RoboDK station: Implementación.rdk

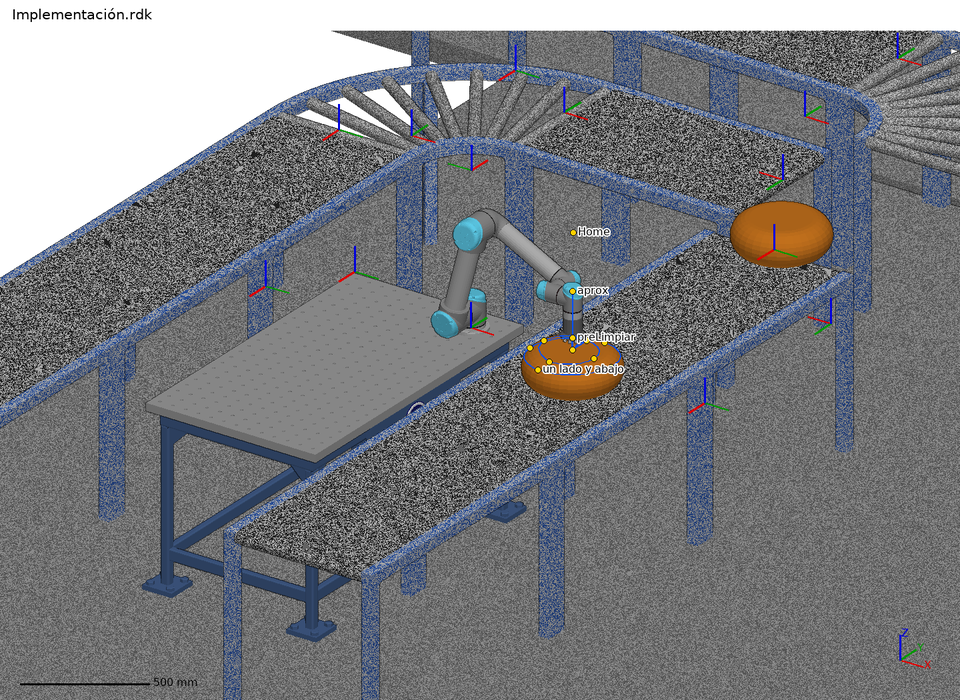
[picture v0: the station drawn from its stored meshes, robots at their saved joint values, targets as dots, program paths as lines]
Station Implementación (saved by RoboDK 5.8.0). Poses are relative to the parent item; angles as X-Y-Z fixed-axis rotations.
  - object Base UR20e at (0, 0, 0) mm, size 250 x 250 x 500 mm, geometry from LayOut general robodk v7 3.step
  - object Suelo at (0, 0, 0) mm, size 13800 x 12750 x 101 mm, geometry from LayOut general robodk v7.step
  - object Estater at (0, 0, 0) mm, size 1550 x 550 x 2250 mm, geometry from LayOut general robodk v7 2.step
  - frame Esquina implantación at (-4000, -50, 1) mm, rotated rx 0 ry 0 rz -90 deg
    - frame mesaRobots at (3150, 1450, 800) mm
      - object mesa at (350, 400, 0) mm, size 1420 x 820 x 800 mm, geometry from Table-1400x800x800mm.sld
      - object keso at (250, 1075, -50) mm, size 400 x 400 x 150 mm, geometry from Queso v10.step
      - frame UR5 Base at (150, 650, 0) mm, rotated rx 0 ry 0 rz 90 deg
        - robot UR5: 6 axes
            modified DH rows (alpha deg, a mm, theta deg, d mm): 0, 0, 0, 89.2; 90, 0, 180, 0; 0, 425, 0, 0; 0, 392, 0, 109.3; -90, 0, 0, 94.75; 90, 0, 180, 82.5
            joint limits [-360, -360, -360, -360, -360, -360] to [360, 360, 360, 360, 360, 360]; home [0, -90, -90, 0, 90, 0]; saved at [0.97, -104.431, -103.116, -62.453, 90, 0.97]
          - tool HerramientaCepillo v3 v3, TCP at (0, 0, 87) mm, size 103 x 102.7 x 101.3 mm, geometry from HerramientaCepillo v3 v3.step
        - target Home (Cartesian target) at (561.5, -109.3, 608.95) mm, rotated rx -90 ry 0 rz -90 deg; joints [0, -90, -90, 0, 90, 0] of UR5
        - target aprox (Cartesian target) at (550, -100, 350) mm, rotated rx 180 ry 0 rz -90 deg; joints [0.97, -98.334, -80.235, -91.431, 90, 0.97] of UR5
        - target preLimpiar (Cartesian target) at (550, -100, 150) mm, rotated rx 180 ry 0 rz -90 deg; joints [158.42, -51.501, -293.37, -285.129, 90, 158.42] of UR5
        - target contactoQueso (Cartesian target) at (550, -100, 100) mm, rotated rx 180 ry 0 rz -90 deg; joints [0.97, -108.044, -106.77, -55.186, 90, 0.97] of UR5
        - target cerca y abajo (Cartesian target) at (362.36, -117.41, 62.97) mm, rotated rx -122.07 ry 2.25 rz -86.41 deg; joints [-5.256, -118.006, -154.949, 60.494, 98.681, -2.826] of UR5
        - target un lado y abajo (Cartesian target) at (510.77, -278.06, 72.55) mm, rotated rx -157.33 ry 40.11 rz -72.05 deg; joints [-29.262, -119.839, -98.457, -65.594, 133.363, -44.391] of UR5
        - target lejos y abajo (Cartesian target) at (730.3, -97.43, 74.87) mm, rotated rx 141.57 ry 25.71 rz -56.33 deg; joints [1.508, -156.051, -23.971, -135.034, 87.527, -40.229] of UR5
        - target otro lado y abajo (Cartesian target) at (570.65, 88.54, 61.08) mm, rotated rx 122.05 ry -0.47 rz -5.3 deg; joints [31.697, -122.988, -92.801, -97.883, 47.184, -34.887] of UR5
        - target cerca (Cartesian target) at (413.04, -94.57, 98.6) mm, rotated rx -179.97 ry -6.45 rz -5.3 deg; joints [2.396, -90.043, -131.065, -42.492, 89.171, -82.352] of UR5
        - target un lado (Cartesian target) at (536.77, -235.76, 98.66) mm, rotated rx -173.55 ry -0.05 rz -4.57 deg; joints [-14.828, -112.038, -101.09, -57.978, 96.358, -100.319] of UR5
        - target lejos (Cartesian target) at (662.53, -118.59, 100) mm, rotated rx 180 ry 0 rz -4.57 deg; joints [-0.803, -121.52, -86.144, -62.337, 90, -86.229] of UR5
        - target otro lado (Cartesian target) at (550.01, -2.99, 100) mm, rotated rx 180 ry 0 rz -4.57 deg; joints [11.151, -106.981, -108.256, -54.763, 90, -74.276] of UR5
    - frame Recta1 at (700, 0, 0) mm, rotated rx 0 ry 0 rz 90 deg
      - robot MecanismoCinta1: 1 axes
          modified DH rows (alpha deg, a mm, theta deg, d mm): 0, 0, 0, 0 linear
          base shift (0, 0, 750) mm, rotated rx 0 ry 90 rz 0 deg
          joint limits [0] to [2030]; home [0]; saved at [0]
        - frame objetoSinta at (0, 325, 0) mm
    - frame Curva1 at (950, 2030, 750) mm, rotated rx 0 ry 0 rz 90 deg
      - robot MecanismoCurva1: 1 axes
          modified DH rows (alpha deg, a mm, theta deg, d mm): 0, 0, 0, 0
          joint limits [-90] to [0]; home [0]; saved at [0]
        - frame objeito at (0, 625, 0) mm
      - object Curva 1 at (0, 0, -750) mm, size 980 x 980 x 750 mm, geometry from Curva v7.step
    - frame Recta2 at (1980, 2280, 0) mm
      - robot MecanismoCinta2: 1 axes
          modified DH rows (alpha deg, a mm, theta deg, d mm): 0, 0, 0, 0 linear
          base shift (0, 0, 750) mm, rotated rx 0 ry 90 rz 0 deg
          joint limits [0] to [3300]; home [0]; saved at [0]
        - frame objeto at (0, 325, 0) mm
          - object keso at (0, -90, 0) mm, size 400 x 400 x 150 mm, geometry from Queso v10.step
    - frame RectaBandeja1 at (1130, 2280, 0) mm, rotated rx 0 ry 0 rz -90 deg
      - robot MecanismoCintaB1: 1 axes
          modified DH rows (alpha deg, a mm, theta deg, d mm): 0, 0, 0, 0 linear
          base shift (0, 0, 750) mm, rotated rx 0 ry 90 rz 0 deg
          joint limits [0] to [1030]; home [0]; saved at [0]
        - frame Objeto at (0, 325, 0) mm
    - frame CurvaBandeja1 at (2080, 1250, 750) mm, rotated rx 0 ry 0 rz 180 deg
      - robot MecanismoCurvaB1: 1 axes
          modified DH rows (alpha deg, a mm, theta deg, d mm): 0, 0, 0, 0
          joint limits [-90] to [0]; home [0]; saved at [-90]
        - frame objeito at (0, 625, 0) mm
      - object CurvaB1 at (0, 0, -750) mm, size 980 x 980 x 750 mm, geometry from Curva v7.step
    - frame RectaBandeja2 at (2110, 300, 0) mm
      - robot MecanismoCintaB2: 1 axes
          modified DH rows (alpha deg, a mm, theta deg, d mm): 0, 0, 0, 0 linear
          base shift (0, 0, 750) mm, rotated rx 0 ry 90 rz 0 deg
          joint limits [-30] to [5030]; home [0]; saved at [-30]
        - frame Objeto at (0, 325, 0) mm
    - frame CurvaBandeja2 at (7140, 1250, 750) mm, rotated rx 0 ry 0 rz -90 deg
      - robot MecanismoCurvaB1: 1 axes
          modified DH rows (alpha deg, a mm, theta deg, d mm): 0, 0, 0, 0
          joint limits [-90] to [0]; home [0]; saved at [-90]
        - frame objeito at (0, 625, 0) mm
      - object CurvaB1 at (0, 0, -750) mm, size 980 x 980 x 750 mm, geometry from Curva v7.step
    - frame RectaBandeja3 at (8090, 1280, 0) mm, rotated rx 0 ry 0 rz 90 deg
      - robot MecanismoCintaB2: 1 axes
          modified DH rows (alpha deg, a mm, theta deg, d mm): 0, 0, 0, 0 linear
          base shift (0, 0, 750) mm, rotated rx 0 ry 90 rz 0 deg
          joint limits [-30] to [5030]; home [0]; saved at [-30]
        - frame Objeto at (0, 325, 0) mm
    - frame CurvaBandeja3 at (7140, 6310, 750) mm
      - robot MecanismoCurvaB1: 1 axes
          modified DH rows (alpha deg, a mm, theta deg, d mm): 0, 0, 0, 0
          joint limits [-90] to [0]; home [0]; saved at [-90]
        - frame objeito at (0, 625, 0) mm
      - object CurvaB1 at (0, 0, -750) mm, size 980 x 980 x 750 mm, geometry from Curva v7.step
    - frame RectaBandeja4 at (7110, 7260, 0) mm, rotated rx 0 ry 0 rz 180 deg
      - robot MecanismoCintaB2: 1 axes
          modified DH rows (alpha deg, a mm, theta deg, d mm): 0, 0, 0, 0 linear
          base shift (0, 0, 750) mm, rotated rx 0 ry 90 rz 0 deg
          joint limits [-30] to [5030]; home [0]; saved at [-30]
        - frame Objeto at (0, 325, 0) mm
    - frame CurvaBandeja4 at (2080, 6310, 750) mm, rotated rx 0 ry 0 rz 90 deg
      - robot MecanismoCurvaB1: 1 axes
          modified DH rows (alpha deg, a mm, theta deg, d mm): 0, 0, 0, 0
          joint limits [-90] to [0]; home [0]; saved at [-90]
        - frame objeito at (0, 625, 0) mm
      - object CurvaB1 at (0, 0, -750) mm, size 980 x 980 x 750 mm, geometry from Curva v7.step
  - program LimpiarQueso (13 instructions, listed below)
  - folder Resets
    - Python program ResetCinta1 (listed below)
    - Python program ResetCurva1 (listed below)
    - Python program ResetCinta2 (listed below)
    - Python program ResetCintaB1 (listed below)
    - Python program ResetCurvaB1 (listed below)
    - Python program ResetCintaB2 (listed below)
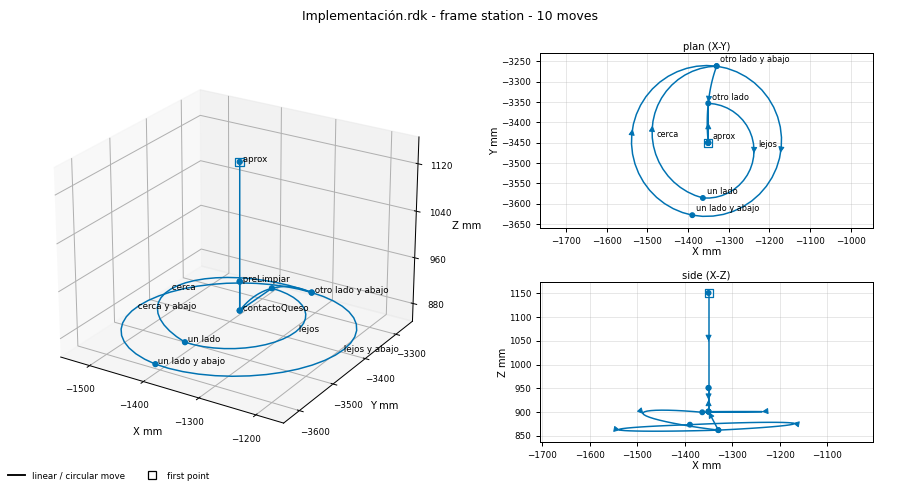
[picture p0: tool path of Implementación.rdk in frame station, 10 of 10 moves have a stored position in this frame; points joined in program order, loops and branches not executed]

--- program LimpiarQueso (robot UR5) ---
  Establecer velocidad (50.0 mm/s)
  Est. Ref.: UR5 Base
  Est. herr: HerramientaCepillo v3 v3
  MoveJ (aprox)
  MoveL (preLimpiar)
  MoveL (contactoQueso)
  MoveL (Target 12) -> target otro lado
  MoveC (Target 11, Target 10) -> target lejos -> target un lado
  MoveC (Target 9, Target 8) -> target cerca -> target otro lado y abajo
  MoveC (Target 7, Target 6) -> target lejos y abajo -> target un lado y abajo
  MoveC (Target 5, Target 8) -> target cerca y abajo -> target otro lado y abajo
  MoveC (Target 12, contactoQueso) -> target otro lado
  MoveL (preLimpiar)

--- Python program ResetCinta1 ---
from robodk.robolink import *  # Importamos la API de RoboDK
from robodk.robomath import *  # Importamos las herramientas matemáticas de RoboDK

# Conectarse al servidor de RoboDK
RDK = Robolink()

# Obtener el mecanismo de la cinta transportadora
cinta = RDK.Item('MecanismoCinta1', ITEM_TYPE_ROBOT)

if not cinta.Valid():
    RDK.ShowMessage("Error: No se encontró un mecanismo llamado 'MecanismoCinta1'.")
    exit()

# Definir las juntas iniciales (reset a 0)
juntas_iniciales = [0]  # Suponemos que la cinta tiene una sola articulación

# Establecer las juntas directamente sin movimiento
cinta.setJoints(juntas_iniciales)

--- Python program ResetCurva1 ---
from robodk.robolink import *  # Importamos la API de RoboDK
from robodk.robomath import *  # Importamos las herramientas matemáticas de RoboDK

# Conectarse al servidor de RoboDK
RDK = Robolink()

# Obtener el mecanismo de la cinta transportadora
cinta = RDK.Item('MecanismoCurva1', ITEM_TYPE_ROBOT)

if not cinta.Valid():
    RDK.ShowMessage("Error: No se encontró un mecanismo llamado 'MecanismoCurva1'.")
    exit()

# Definir las juntas iniciales (reset a 0)
juntas_iniciales = [0]  # Suponemos que la cinta tiene una sola articulación

# Establecer las juntas directamente sin movimiento
cinta.setJoints(juntas_iniciales)

--- Python program ResetCinta2 ---
from robodk.robolink import *  # Importamos la API de RoboDK
from robodk.robomath import *  # Importamos las herramientas matemáticas de RoboDK

# Conectarse al servidor de RoboDK
RDK = Robolink()

# Obtener el mecanismo de la cinta transportadora
cinta = RDK.Item('MecanismoCinta2', ITEM_TYPE_ROBOT)

if not cinta.Valid():
    RDK.ShowMessage("Error: No se encontró un mecanismo llamado 'MecanismoCinta2'.")
    exit()

# Definir las juntas iniciales (reset a 0)
juntas_iniciales = [0]  # Suponemos que la cinta tiene una sola articulación

# Establecer las juntas directamente sin movimiento
cinta.setJoints(juntas_iniciales)

--- Python program ResetCintaB1 ---
from robodk.robolink import *  # Importamos la API de RoboDK
from robodk.robomath import *  # Importamos las herramientas matemáticas de RoboDK

# Conectarse al servidor de RoboDK
RDK = Robolink()

# Obtener el mecanismo de la cinta transportadora
cinta = RDK.Item('MecanismoCintaB1', ITEM_TYPE_ROBOT)

if not cinta.Valid():
    RDK.ShowMessage("Error: No se encontró un mecanismo llamado 'MecanismoCintaB1'.")
    exit()

# Definir las juntas iniciales (reset a 0)
juntas_iniciales = [0]  # Suponemos que la cinta tiene una sola articulación

# Establecer las juntas directamente sin movimiento
cinta.setJoints(juntas_iniciales)

--- Python program ResetCurvaB1 ---
from robodk.robolink import *  # Importamos la API de RoboDK
from robodk.robomath import *  # Importamos las herramientas matemáticas de RoboDK

# Conectarse al servidor de RoboDK
RDK = Robolink()

# Obtener el mecanismo de la cinta transportadora
cinta = RDK.Item('MecanismoCurvaB1', ITEM_TYPE_ROBOT)

if not cinta.Valid():
    RDK.ShowMessage("Error: No se encontró un mecanismo llamado 'MecanismoCurvaB1'.")
    exit()

# Definir las juntas iniciales (reset a 0)
juntas_iniciales = [-90]  # Suponemos que la cinta tiene una sola articulación

# Establecer las juntas directamente sin movimiento
cinta.setJoints(juntas_iniciales)

--- Python program ResetCintaB2 ---
from robodk.robolink import *  # Importamos la API de RoboDK
from robodk.robomath import *  # Importamos las herramientas matemáticas de RoboDK

# Conectarse al servidor de RoboDK
RDK = Robolink()

# Obtener el mecanismo de la cinta transportadora
cinta = RDK.Item('MecanismoCintaB2', ITEM_TYPE_ROBOT)

if not cinta.Valid():
    RDK.ShowMessage("Error: No se encontró un mecanismo llamado 'MecanismoCintaB2'.")
    exit()

# Definir las juntas iniciales (reset a 0)
juntas_iniciales = [-30]  # Suponemos que la cinta tiene una sola articulación

# Establecer las juntas directamente sin movimiento
cinta.setJoints(juntas_iniciales)
